// TIA Portal V19 export
TYPE "dtSupply"
   STRUCT
      setAvailPumps { S7_SetPoint := 'True'} : Array[0..3] of Bool;
      loadAvailPumps : Array[0..3] of Bool;
      availPumps : Array[0..2] of Bool;
      loadBtn : Bool := FALSE;
      pressureSP { S7_SetPoint := 'True'} : Real;
      hhPressureAlm : Real;
      highFlow { S7_SetPoint := 'True'} : Real;
      lowFlow { S7_SetPoint := 'True'} : Real;
      zChangeThr : Real := 0.5;
      zChangeDelay { S7_SetPoint := 'True'} : Time;
      PumpInterval : Time := T#10m;
      zoneChangeOP : Real := 95.0;
      overlapDelay : Time := T#60S;
      downgradeDelay : Time := T#10s;
      chLead : Int;
      enRotation : Bool;
      stageUp { S7_SetPoint := 'True'} : "dtStageUp";
      stageDown : Array[0..3] of "dtStageDown";
   END_STRUCT;
   // setAvailPumps[0..2] := 0;
END_TYPE
